TYPE S2_location:
    (S2_A, S2_B);
END_TYPE

(* stored: ProductVersion 3.1.0.18, Version 1.1.0.1 *)
